// TIA Portal V20 export
VAR_GLOBAL   // PLC tag table "Approach_type"
   send AT %M1.0 : Bool;
   testmqtt AT %M1.1 : Bool;
END_VAR
VAR_GLOBAL CONSTANT   // user constants
   XX : Int := 1;
   YY : Int := 2;
   ZZ : Int := 3;
   XZ : Int := 4;
   ZX : Int := 5;
   YZ : Int := 6;
   ZY : Int := 7;
   XY : Int := 8;
   YX : Int := 9;
END_VAR
